TYPE T_RecipeId : STRING(20); END_TYPE

(* stored: Version 1.1.0.1, ProductVersion 3.1.4024.15
   DUT T_RecipeId: Id {7fe15058-6828-4f35-b62b-24b1b68d08ad} *)
